Fanuc KAREL source: w_d_defg.kl

PROGRAM w_d_defg
%NOLOCKGROUP
%DEFGROUP = 2
VAR
  p : POSITION
  r : REAL
BEGIN
  WITH $SPEED = 500 MOVE TO p
  WITH $SPEED = r, $MOTYPE = LINEAR MOVE TO p
END w_d_defg
